PROGRAM SafetyInterface_MtrCntrl055
VAR
	
	pMtrRunning: POINTER TO ConvMtrRunningPuck;
	pSafety: POINTER TO Plc2PlcDataSafetyPuckConv;
	
// Stn055_05_StnMain.MotorCtrl
// Update the station and naming to first motor the station is controlling	
//	StartIndexThisMotor to sequential number that allows two motors at a time "per enclosure"  to start (see max index limit above)
//	hoMtrName to appropriate enclosure and motor number
//	gMtrRunning.EncXXXMtrYYY to appropriate member of the running DUT

// Call to motor control function block for each main line motor	
// Blue Storage - Enc51:  3,4,5,6  Enc61: 6  Enc62: 8,9
// Red Storage  - Enc51:  2 Enc61: 5 Enc52: 3,4,6,7
// Grn Storage  - Enc51:  1 Enc61: 1,2,4  Enc62: 1,2
	{attribute 'TcLinkToOSO' := '	
		.Enc051Mtr01.iDisconnectOk  :=  <0,1,2>TIIB[N13S00 (AL1332)]^N13S01 (AL2341)^TxPDO^input byte 3;
		.Enc051Mtr02.iDisconnectOk  :=  <0,1,3>TIIB[N13S00 (AL1332)]^N13S01 (AL2341)^TxPDO^input byte 1;
		.Enc051Mtr03.iDisconnectOk  :=  <0,1,4>TIIB[N12S00 (AL1332)]^N12S03 (AL2341)^TxPDO^input byte 3;
		.Enc051Mtr04.iDisconnectOk  :=  <0,1,4>TIIB[N12S00 (AL1332)]^N12S05 (AL2341)^TxPDO^input byte 1;
		.Enc051Mtr05.iDisconnectOk  :=  <0,1,4>TIIB[N12S00 (AL1332)]^N12S05 (AL2341)^TxPDO^input byte 3;
		.Enc051Mtr06.iDisconnectOk  :=  <0,1,3>TIIB[N13S00 (AL1332)]^N13S01 (AL2341)^TxPDO^input byte 3;
		.Enc061Mtr01.iDisconnectOk  :=  <0,1,4>TIIB[N66S00 (AL1332)]^N66S03 (AL2341)^TxPDO^input byte 3;
		.Enc061Mtr02.iDisconnectOk  :=  <0,1,4>TIIB[N67S00 (AL1332)]^N67S03 (AL2341)^TxPDO^input byte 3;
		.Enc061Mtr03.iDisconnectOk  :=  <0,1,4>TIIB[N67S00 (AL1332)]^N67S05 (AL2341)^TxPDO^input byte 1; 
		.Enc061Mtr04.iDisconnectOk  :=  <0,1,4>TIIB[N67S00 (AL1332)]^N67S05 (AL2341)^TxPDO^input byte 3;
		.Enc061Mtr05.iDisconnectOk  :=  <0,1,4>TIIB[N66S00 (AL1332)]^N66S07 (AL2341)^TxPDO^input byte 1;
		.Enc061Mtr06.iDisconnectOk  :=  <0,1,4>TIIB[N66S00 (AL1332)]^N66S07 (AL2341)^TxPDO^input byte 3;
		.Enc062Mtr01.iDisconnectOk :=  <0,1,4>TIIB[N71S00 (AL1332)]^N71S01 (AL2341)^TxPDO^input byte 3;
		.Enc062Mtr02.iDisconnectOk :=  <0,1,4>TIIB[N73S00 (AL1332)]^N73S01 (AL2341)^TxPDO^input byte 1;
		.Enc062Mtr03.iDisconnectOk :=  <0,1,4>TIIB[N71S00 (AL1332)]^N71S03 (AL2341)^TxPDO^input byte 3;
		.Enc062Mtr04.iDisconnectOk :=  <0,1,4>TIIB[N72S00 (AL1332)]^N72S03 (AL2341)^TxPDO^input byte 3;
		.Enc062Mtr05.iDisconnectOk :=  <0,1,4>TIIB[N72S00 (AL1332)]^N72S05 (AL2341)^TxPDO^input byte 1;
		.Enc062Mtr06.iDisconnectOk :=  <0,1,4>TIIB[N71S00 (AL1332)]^N71S05 (AL2341)^TxPDO^input byte 1;
		.Enc062Mtr07.iDisconnectOk :=  <0,1,4>TIIB[N73S00 (AL1332)]^N73S05 (AL2341)^TxPDO^input byte 1;
		.Enc062Mtr08.iDisconnectOk :=  <0,1,4>TIIB[N71S00 (AL1332)]^N71S05 (AL2341)^TxPDO^input byte 3;
		.Enc062Mtr09.iDisconnectOk :=  <0,1,4>TIIB[N73S00 (AL1332)]^N73S05 (AL2341)^TxPDO^input byte 3'}
	{attribute 'TcLinkTo' := '	
		.Enc051Mtr01.iOverloadTripped  := TIIB[N10S06 (EL1008)]^Channel 6^Input;
		.Enc051Mtr02.iOverloadTripped  := TIIB[N10S06 (EL1008)]^Channel 8^Input;
		.Enc051Mtr03.iOverloadTripped  := TIIB[N10S07 (EL1008)]^Channel 2^Input;
		.Enc051Mtr04.iOverloadTripped  := TIIB[N10S07 (EL1008)]^Channel 4^Input;
		.Enc051Mtr05.iOverloadTripped  := TIIB[N10S07 (EL1008)]^Channel 6^Input;
		.Enc051Mtr06.iOverloadTripped  := TIIB[N10S07 (EL1008)]^Channel 8^Input;
		.Enc061Mtr01.iOverloadTripped  := TIIB[N65S06 (EL1008)]^Channel 6^Input;
		.Enc061Mtr02.iOverloadTripped  := TIIB[N65S06 (EL1008)]^Channel 8^Input;
		.Enc061Mtr03.iOverloadTripped  := TIIB[N65S07 (EL1008)]^Channel 2^Input;
		.Enc061Mtr04.iOverloadTripped  := TIIB[N65S07 (EL1008)]^Channel 6^Input;
		.Enc061Mtr05.iOverloadTripped  := TIIB[N65S07 (EL1008)]^Channel 8^Input;
		.Enc061Mtr06.iOverloadTripped  := TIIB[N65S08 (EL1008)]^Channel 2^Input;
		.Enc062Mtr01.iOverloadTripped := TIIB[N70S06 (EL1008)]^Channel 6^Input;
		.Enc062Mtr02.iOverloadTripped := TIIB[N70S06 (EL1008)]^Channel 8^Input;
		.Enc062Mtr03.iOverloadTripped := TIIB[N70S07 (EL1008)]^Channel 2^Input;
		.Enc062Mtr04.iOverloadTripped := TIIB[N70S07 (EL1008)]^Channel 4^Input;
		.Enc062Mtr05.iOverloadTripped := TIIB[N70S07 (EL1008)]^Channel 6^Input;
		.Enc062Mtr06.iOverloadTripped := TIIB[N70S07 (EL1008)]^Channel 8^Input;
		.Enc062Mtr07.iOverloadTripped := TIIB[N70S08 (EL1008)]^Channel 2^Input;
		.Enc062Mtr08.iOverloadTripped := TIIB[N70S08 (EL1008)]^Channel 4^Input;
		.Enc062Mtr09.iOverloadTripped := TIIB[N70S08 (EL1008)]^Channel 6^Input;
		.Enc051Mtr01.iRunning  := TIIB[N10S06 (EL1008)]^Channel 5^Input;
		.Enc051Mtr02.iRunning  := TIIB[N10S06 (EL1008)]^Channel 7^Input;
		.Enc051Mtr03.iRunning  := TIIB[N10S07 (EL1008)]^Channel 1^Input;
		.Enc051Mtr04.iRunning  := TIIB[N10S07 (EL1008)]^Channel 3^Input;
		.Enc051Mtr05.iRunning  := TIIB[N10S07 (EL1008)]^Channel 5^Input;
		.Enc051Mtr06.iRunning  := TIIB[N10S07 (EL1008)]^Channel 7^Input;
		.Enc061Mtr01.iRunning  := TIIB[N65S06 (EL1008)]^Channel 5^Input;
		.Enc061Mtr02.iRunning  := TIIB[N65S06 (EL1008)]^Channel 7^Input;
		.Enc061Mtr03.iRunning  := TIIB[N65S07 (EL1008)]^Channel 1^Input;
		.Enc061Mtr04.iRunning  := TIIB[N65S07 (EL1008)]^Channel 5^Input;
		.Enc061Mtr05.iRunning  := TIIB[N65S07 (EL1008)]^Channel 7^Input;
		.Enc061Mtr06.iRunning  := TIIB[N65S08 (EL1008)]^Channel 1^Input;
		.Enc062Mtr01.iRunning := TIIB[N70S06 (EL1008)]^Channel 5^Input;
		.Enc062Mtr02.iRunning := TIIB[N70S06 (EL1008)]^Channel 7^Input;
		.Enc062Mtr03.iRunning := TIIB[N70S07 (EL1008)]^Channel 1^Input;
		.Enc062Mtr04.iRunning := TIIB[N70S07 (EL1008)]^Channel 3^Input;
		.Enc062Mtr05.iRunning := TIIB[N70S07 (EL1008)]^Channel 5^Input;
		.Enc062Mtr06.iRunning := TIIB[N70S07 (EL1008)]^Channel 7^Input;
		.Enc062Mtr07.iRunning := TIIB[N70S08 (EL1008)]^Channel 1^Input;
		.Enc062Mtr08.iRunning := TIIB[N70S08 (EL1008)]^Channel 3^Input;
		.Enc062Mtr09.iRunning := TIIB[N70S08 (EL1008)]^Channel 5^Input;
		.Enc051Mtr01.oRun  := TIIB[N10S12 (EL2008)]^Channel 4^Output;
		.Enc051Mtr02.oRun  := TIIB[N10S12 (EL2008)]^Channel 5^Output;
		.Enc051Mtr03.oRun  := TIIB[N10S12 (EL2008)]^Channel 6^Output;
		.Enc051Mtr04.oRun  := TIIB[N10S12 (EL2008)]^Channel 7^Output;
		.Enc051Mtr05.oRun  := TIIB[N10S12 (EL2008)]^Channel 8^Output;
		.Enc051Mtr06.oRun  := TIIB[N10S13 (EL2008)]^Channel 1^Output;
		.Enc061Mtr01.oRun  := TIIB[N65S12 (EL2008)]^Channel 5^Output;
		.Enc061Mtr02.oRun  := TIIB[N65S12 (EL2008)]^Channel 6^Output;
		.Enc061Mtr03.oRun  := TIIB[N65S12 (EL2008)]^Channel 7^Output;
		.Enc061Mtr04.oRun  := TIIB[N65S13 (EL2008)]^Channel 1^Output;
		.Enc061Mtr05.oRun  := TIIB[N65S13 (EL2008)]^Channel 2^Output;
		.Enc061Mtr06.oRun  := TIIB[N65S13 (EL2008)]^Channel 3^Output;
		.Enc062Mtr01.oRun := TIIB[N70S12 (EL2008)]^Channel 5^Output;
		.Enc062Mtr02.oRun := TIIB[N70S12 (EL2008)]^Channel 6^Output;
		.Enc062Mtr03.oRun := TIIB[N70S12 (EL2008)]^Channel 7^Output;
		.Enc062Mtr04.oRun := TIIB[N70S12 (EL2008)]^Channel 8^Output;
		.Enc062Mtr05.oRun := TIIB[N70S13 (EL2008)]^Channel 1^Output;
		.Enc062Mtr06.oRun := TIIB[N70S13 (EL2008)]^Channel 2^Output;
		.Enc062Mtr07.oRun := TIIB[N70S13 (EL2008)]^Channel 3^Output;
		.Enc062Mtr08.oRun := TIIB[N70S13 (EL2008)]^Channel 4^Output;
		.Enc062Mtr09.oRun := TIIB[N70S13 (EL2008)]^Channel 5^Output'}
	MtrCtrls: ConvMtrCtrlsPuck;

	MtrNOKtoRun : BOOL;	
	cntMotorStartIndex: DINT;	
	tmrMotorStartIndex: TON;

END_VAR
VAR CONSTANT	
	
	cMaxMotorStartIndex :DINT := 9;  //If starting pairs of motors  adjust to max number of motors "per enclosure" /2
	
END_VAR

pMtrRunning := ADR(gProduced_SafetyInterfaceConv.MtrRunning);
pSafety := ADR(gProduced_SafetyInterfaceConv);

//Create sequenced motor start index - to prevent inrush overloads at time of motor start		
tmrMotorStartIndex(IN:=NOT tmrMotorStartIndex.Q,PT:=T#300ms);		
IF tmrMotorStartIndex.Q THEN 		
	cntMotorStartIndex := cntMotorStartIndex + 1;	
	IF cntMotorStartIndex > cMaxMotorStartIndex THEN 	
		cntMotorStartIndex := 1;
	END_IF	
END_IF	

// Call action code block that does call for each main line motor		
MotorCtrl();

//distibute the incoming stn data (consumed data from stn) to single produced outgoing to all stns
//MEMCPY(ADR(gProduced_SafetyInterfaceConv.gMtrRunningStn051), ADR(gMtrRunning), SizeOf(gProduced_SafetyInterfaceConv.gMtrRunningStn051));

ACTION MotorCtrl:
// Stn055_05_StnMain.MotorCtrl
// Update the station and naming to first motor the station is controlling	
//	StartIndexThisMotor to sequential number that allows two motors at a time "per enclosure"  to start (see max index limit above)
//	hoMtrName to appropriate enclosure and motor number
//	gMtrRunning.EncXXXMtrYYY to appropriate member of the running DUT

//TODO remove when switching to real motor control
//gMainConvRunning := TRUE;

// Call to motor control function block for each main line motor	
// Blue Storage - Enc51:  3,4,5,6  Enc61: 6  	Enc62: 8,9
// Red Storage  - Enc51:  2 	Enc61: 5 		Enc62: 3,4,5,6,7
// Grn Storage  - Enc51:  1 	Enc61: 1,2,3,4  Enc62: 1,2

MtrCtrls.Enc051Mtr01(	
	CycleAuto := gConsumed_Stn055ToSafetyInterface.CycleAuto,
	CycleReset := gConsumed_Stn055ToSafetyInterface.CycleReset,
	NOKtoRun := pSafety^.Enc051.iEstopRlyTripped,	
//	NOKtoRun := pSafety^.Enc051.iEstopRlyTripped OR 
//		NOT gConsumed_Stn055ToSafetyInterface.Stn055PLCData[2].3 OR 
//		NOT gConsumed_Stn055ToSafetyInterface_OK,		
	StartIndexThisMotor := 1,
	StartIndexCurrent := cntMotorStartIndex,
	hoMtrName := 'Enc051-Mtr1',
	MtrRunning => pMtrRunning^.Enc051Mtr01);

MtrCtrls.Enc051Mtr02(	
	CycleAuto := gConsumed_Stn055ToSafetyInterface.CycleAuto,
	CycleReset := gConsumed_Stn055ToSafetyInterface.CycleReset,
	NOKtoRun := pSafety^.Enc051.iEstopRlyTripped,	
//	NOKtoRun := pSafety^.Enc051.iEstopRlyTripped OR 
//		NOT gConsumed_Stn055ToSafetyInterface.Stn055PLCData[2].3 OR 
//		NOT gConsumed_Stn055ToSafetyInterface_OK,		
	StartIndexThisMotor := 1,
	StartIndexCurrent := cntMotorStartIndex,
	hoMtrName := 'Enc051-Mtr2',
	MtrRunning => pMtrRunning^.Enc051Mtr02);

MtrCtrls.Enc051Mtr03(	
	CycleAuto := gConsumed_Stn055ToSafetyInterface.CycleAuto,
	CycleReset := gConsumed_Stn055ToSafetyInterface.CycleReset,
	NOKtoRun := pSafety^.Enc051.iEstopRlyTripped,	
//	NOKtoRun := pSafety^.Enc051.iEstopRlyTripped OR 
//		NOT gConsumed_Stn055ToSafetyInterface.Stn055PLCData[2].3 OR 
//		NOT gConsumed_Stn055ToSafetyInterface_OK,		
	StartIndexThisMotor := 2,
	StartIndexCurrent := cntMotorStartIndex,
	hoMtrName := 'Enc051-Mtr3',
	MtrRunning => pMtrRunning^.Enc051Mtr03);

MtrCtrls.Enc051Mtr04(	
	CycleAuto := gConsumed_Stn055ToSafetyInterface.CycleAuto,
	CycleReset := gConsumed_Stn055ToSafetyInterface.CycleReset,
	NOKtoRun := pSafety^.Enc051.iEstopRlyTripped,	
//	NOKtoRun := pSafety^.Enc051.iEstopRlyTripped OR 
//		NOT gConsumed_Stn055ToSafetyInterface.Stn055PLCData[2].3 OR 
//		NOT gConsumed_Stn055ToSafetyInterface_OK,		
	StartIndexThisMotor := 2,
	StartIndexCurrent := cntMotorStartIndex,
	hoMtrName := 'Enc051-Mtr4',
	MtrRunning => pMtrRunning^.Enc051Mtr04);

MtrCtrls.Enc051Mtr05(	
	CycleAuto := gConsumed_Stn055ToSafetyInterface.CycleAuto,
	CycleReset := gConsumed_Stn055ToSafetyInterface.CycleReset,
	NOKtoRun := pSafety^.Enc051.iEstopRlyTripped,	
//	NOKtoRun := pSafety^.Enc051.iEstopRlyTripped OR 
//		NOT gConsumed_Stn055ToSafetyInterface.Stn055PLCData[2].3 OR 
//		NOT gConsumed_Stn055ToSafetyInterface_OK,		
	StartIndexThisMotor := 3,
	StartIndexCurrent := cntMotorStartIndex,
	hoMtrName := 'Enc051-Mtr5',
	MtrRunning => pMtrRunning^.Enc051Mtr05);

MtrCtrls.Enc051Mtr06(	
	CycleAuto := gConsumed_Stn055ToSafetyInterface.CycleAuto,
	CycleReset := gConsumed_Stn055ToSafetyInterface.CycleReset,
	NOKtoRun := pSafety^.Enc051.iEstopRlyTripped,	
//	NOKtoRun := pSafety^.Enc051.iEstopRlyTripped OR 
//		NOT gConsumed_Stn055ToSafetyInterface.Stn055PLCData[2].3 OR 
//		NOT gConsumed_Stn055ToSafetyInterface_OK,		
	StartIndexThisMotor := 3,
	StartIndexCurrent := cntMotorStartIndex,
	hoMtrName := 'Enc051-Mtr6',
	MtrRunning => pMtrRunning^.Enc051Mtr06);

MtrCtrls.Enc061Mtr01(	
	CycleAuto := gConsumed_Stn055ToSafetyInterface.CycleAuto,
	CycleReset := gConsumed_Stn055ToSafetyInterface.CycleReset,
	NOKtoRun := pSafety^.Enc061.iEstopRlyTripped,	
//	NOKtoRun := pSafety^.Enc061.iEstopRlyTripped OR 
//		NOT gConsumed_Stn055ToSafetyInterface.Stn055PLCData[2].3 OR 
//		NOT gConsumed_Stn055ToSafetyInterface_OK,		
	StartIndexThisMotor := 4,
	StartIndexCurrent := cntMotorStartIndex,
	hoMtrName := 'Enc061-Mtr1',
	MtrRunning => pMtrRunning^.Enc061Mtr01);

MtrCtrls.Enc061Mtr02(	
	CycleAuto := gConsumed_Stn055ToSafetyInterface.CycleAuto,
	CycleReset := gConsumed_Stn055ToSafetyInterface.CycleReset,
	NOKtoRun := pSafety^.Enc061.iEstopRlyTripped,	
//	NOKtoRun := pSafety^.Enc061.iEstopRlyTripped OR 
//		NOT gConsumed_Stn055ToSafetyInterface.Stn055PLCData[2].3 OR 
//		NOT gConsumed_Stn055ToSafetyInterface_OK,		
	StartIndexThisMotor := 4,
	StartIndexCurrent := cntMotorStartIndex,
	hoMtrName := 'Enc061-Mtr2',
	MtrRunning => pMtrRunning^.Enc061Mtr02);

MtrCtrls.Enc061Mtr03(	
	CycleAuto := gConsumed_Stn055ToSafetyInterface.CycleAuto,
	CycleReset := gConsumed_Stn055ToSafetyInterface.CycleReset,
	NOKtoRun := pSafety^.Enc061.iEstopRlyTripped,	
//	NOKtoRun := pSafety^.Enc061.iEstopRlyTripped OR 
//		NOT gConsumed_Stn055ToSafetyInterface.Stn055PLCData[2].3 OR 
//		NOT gConsumed_Stn055ToSafetyInterface_OK,		
	StartIndexThisMotor := 4,
	StartIndexCurrent := cntMotorStartIndex,
	hoMtrName := 'Enc061-Mtr3',
	MtrRunning => pMtrRunning^.Enc061Mtr03);

MtrCtrls.Enc061Mtr04(	
	CycleAuto := gConsumed_Stn055ToSafetyInterface.CycleAuto,
	CycleReset := gConsumed_Stn055ToSafetyInterface.CycleReset,
	NOKtoRun := pSafety^.Enc061.iEstopRlyTripped,	
//	NOKtoRun := pSafety^.Enc061.iEstopRlyTripped OR 
//		NOT gConsumed_Stn055ToSafetyInterface.Stn055PLCData[2].3 OR 
//		NOT gConsumed_Stn055ToSafetyInterface_OK,		
	StartIndexThisMotor := 5,
	StartIndexCurrent := cntMotorStartIndex,
	hoMtrName := 'Enc061-Mtr4',
	MtrRunning => pMtrRunning^.Enc061Mtr04);

MtrCtrls.Enc061Mtr05(	
	CycleAuto := gConsumed_Stn055ToSafetyInterface.CycleAuto,
	CycleReset := gConsumed_Stn055ToSafetyInterface.CycleReset,
	NOKtoRun := pSafety^.Enc061.iEstopRlyTripped,	
//	NOKtoRun := pSafety^.Enc061.iEstopRlyTripped OR 
//		NOT gConsumed_Stn055ToSafetyInterface.Stn055PLCData[2].3 OR 
//		NOT gConsumed_Stn055ToSafetyInterface_OK,		
	StartIndexThisMotor := 5,
	StartIndexCurrent := cntMotorStartIndex,
	hoMtrName := 'Enc061-Mtr5',
	MtrRunning => pMtrRunning^.Enc061Mtr05);

MtrCtrls.Enc061Mtr06(	
	CycleAuto := gConsumed_Stn055ToSafetyInterface.CycleAuto,
	CycleReset := gConsumed_Stn055ToSafetyInterface.CycleReset,
	NOKtoRun := pSafety^.Enc061.iEstopRlyTripped,	
//	NOKtoRun := pSafety^.Enc061.iEstopRlyTripped OR 
//		NOT gConsumed_Stn055ToSafetyInterface.Stn055PLCData[2].3 OR 
//		NOT gConsumed_Stn055ToSafetyInterface_OK,		
	StartIndexThisMotor := 6,
	StartIndexCurrent := cntMotorStartIndex,
	hoMtrName := 'Enc061-Mtr6',
	MtrRunning => pMtrRunning^.Enc061Mtr06);

MtrCtrls.Enc062Mtr01(	
	CycleAuto := gConsumed_Stn055ToSafetyInterface.CycleAuto,
	CycleReset := gConsumed_Stn055ToSafetyInterface.CycleReset,
	NOKtoRun := pSafety^.Enc062.iEstopRlyTripped,	
//	NOKtoRun := pSafety^.Enc062.iEstopRlyTripped OR 
//		NOT gConsumed_Stn055ToSafetyInterface.Stn055PLCData[2].3 OR 
//		NOT gConsumed_Stn055ToSafetyInterface_OK,		
	StartIndexThisMotor := 6,
	StartIndexCurrent := cntMotorStartIndex,
	hoMtrName := 'Enc062-Mtr1',
	MtrRunning => pMtrRunning^.Enc062Mtr01);

MtrCtrls.Enc062Mtr02(	
	CycleAuto := gConsumed_Stn055ToSafetyInterface.CycleAuto,
	CycleReset := gConsumed_Stn055ToSafetyInterface.CycleReset,
	NOKtoRun := pSafety^.Enc062.iEstopRlyTripped,	
//	NOKtoRun := pSafety^.Enc062.iEstopRlyTripped OR 
//		NOT gConsumed_Stn055ToSafetyInterface.Stn055PLCData[2].3 OR 
//		NOT gConsumed_Stn055ToSafetyInterface_OK,		
	StartIndexThisMotor := 7,
	StartIndexCurrent := cntMotorStartIndex,
	hoMtrName := 'Enc062-Mtr2',
	MtrRunning => pMtrRunning^.Enc062Mtr02);

MtrCtrls.Enc062Mtr03(	
	CycleAuto := gConsumed_Stn055ToSafetyInterface.CycleAuto,
	CycleReset := gConsumed_Stn055ToSafetyInterface.CycleReset,
	NOKtoRun := pSafety^.Enc062.iEstopRlyTripped,	
//	NOKtoRun := pSafety^.Enc062.iEstopRlyTripped OR 
//		NOT gConsumed_Stn055ToSafetyInterface.Stn055PLCData[2].3 OR 
//		NOT gConsumed_Stn055ToSafetyInterface_OK,		
	StartIndexThisMotor := 7,
	StartIndexCurrent := cntMotorStartIndex,
	hoMtrName := 'Enc062-Mtr3',
	MtrRunning => pMtrRunning^.Enc062Mtr03);

MtrCtrls.Enc062Mtr04(	
	CycleAuto := gConsumed_Stn055ToSafetyInterface.CycleAuto,
	CycleReset := gConsumed_Stn055ToSafetyInterface.CycleReset,
	NOKtoRun := pSafety^.Enc062.iEstopRlyTripped,	
//	NOKtoRun := pSafety^.Enc062.iEstopRlyTripped OR 
//		NOT gConsumed_Stn055ToSafetyInterface.Stn055PLCData[2].3 OR 
//		NOT gConsumed_Stn055ToSafetyInterface_OK,		
	StartIndexThisMotor := 8,
	StartIndexCurrent := cntMotorStartIndex,
	hoMtrName := 'Enc062-Mtr4',
	MtrRunning => pMtrRunning^.Enc062Mtr04);

MtrCtrls.Enc062Mtr05(	
	CycleAuto := gConsumed_Stn055ToSafetyInterface.CycleAuto,
	CycleReset := gConsumed_Stn055ToSafetyInterface.CycleReset,
	NOKtoRun := pSafety^.Enc062.iEstopRlyTripped,	
//	NOKtoRun := pSafety^.Enc062.iEstopRlyTripped OR 
//		NOT gConsumed_Stn055ToSafetyInterface.Stn055PLCData[2].3 OR 
//		NOT gConsumed_Stn055ToSafetyInterface_OK,		
	StartIndexThisMotor := 8,
	StartIndexCurrent := cntMotorStartIndex,
	hoMtrName := 'Enc062-Mtr5',
	MtrRunning => pMtrRunning^.Enc062Mtr05);

MtrCtrls.Enc062Mtr06(	
	CycleAuto := gConsumed_Stn055ToSafetyInterface.CycleAuto,
	CycleReset := gConsumed_Stn055ToSafetyInterface.CycleReset,
	NOKtoRun := pSafety^.Enc062.iEstopRlyTripped,	
//	NOKtoRun := pSafety^.Enc062.iEstopRlyTripped OR 
//		NOT gConsumed_Stn055ToSafetyInterface.Stn055PLCData[2].3 OR 
//		NOT gConsumed_Stn055ToSafetyInterface_OK,		
	StartIndexThisMotor := 8,
	StartIndexCurrent := cntMotorStartIndex,
	hoMtrName := 'Enc062-Mtr6',
	MtrRunning => pMtrRunning^.Enc062Mtr06);

MtrCtrls.Enc062Mtr07(	
	CycleAuto := gConsumed_Stn055ToSafetyInterface.CycleAuto,
	CycleReset := gConsumed_Stn055ToSafetyInterface.CycleReset,
	NOKtoRun := pSafety^.Enc062.iEstopRlyTripped,	
//	NOKtoRun := pSafety^.Enc062.iEstopRlyTripped OR 
//		NOT gConsumed_Stn055ToSafetyInterface.Stn055PLCData[2].3 OR 
//		NOT gConsumed_Stn055ToSafetyInterface_OK,		
	StartIndexThisMotor := 9,
	StartIndexCurrent := cntMotorStartIndex,
	hoMtrName := 'Enc062-Mtr7',
	MtrRunning => pMtrRunning^.Enc062Mtr07);

MtrCtrls.Enc062Mtr08(	
	CycleAuto := gConsumed_Stn055ToSafetyInterface.CycleAuto,
	CycleReset := gConsumed_Stn055ToSafetyInterface.CycleReset,
	NOKtoRun := pSafety^.Enc062.iEstopRlyTripped,	
//	NOKtoRun := pSafety^.Enc062.iEstopRlyTripped OR 
//		NOT gConsumed_Stn055ToSafetyInterface.Stn055PLCData[2].3 OR 
//		NOT gConsumed_Stn055ToSafetyInterface_OK,		
	StartIndexThisMotor := 9,
	StartIndexCurrent := cntMotorStartIndex,
	hoMtrName := 'Enc062-Mtr8',
	MtrRunning => pMtrRunning^.Enc062Mtr08);

MtrCtrls.Enc062Mtr09(	
	CycleAuto := gConsumed_Stn055ToSafetyInterface.CycleAuto,
	CycleReset := gConsumed_Stn055ToSafetyInterface.CycleReset,
	NOKtoRun := pSafety^.Enc062.iEstopRlyTripped,	
//	NOKtoRun := pSafety^.Enc062.iEstopRlyTripped OR 
//		NOT gConsumed_Stn055ToSafetyInterface.Stn055PLCData[2].3 OR 
//		NOT gConsumed_Stn055ToSafetyInterface_OK,		
	StartIndexThisMotor := 9,
	StartIndexCurrent := cntMotorStartIndex,
	hoMtrName := 'Enc062-Mtr9',
	MtrRunning => pMtrRunning^.Enc062Mtr09);
	
	
//For each motor that the station needs running information but NOT actually controlling the output… 
//(populate the running bit from the produced consumed logic)

// Populate motor running for motors controlled (outputs linked) by other stations
//gMtrRunning.Enc062Mtr07 := gConsumed_Stn901To902.ScratchPad[10].0;
END_ACTION

END_PROGRAM

(* stored: Version 1.1.0.1, ProductVersion 3.1.4024.6
   POU SafetyInterface_MtrCntrl055: Id {ecea5fe9-41b1-4e7e-8a1a-d5dffb2b1786}, SpecialFunc None
   Action MotorCtrl: Id {da34b849-e349-46d2-b88a-22fcae3641d2} *)
